// TIA Portal V15.1 export
// export: Created 2020-06-12T07:35:47.7568359Z, ExportSetting None, DisplayName Totally Integrated Automation Portal, DisplayVersion V15.1, DisplayName TIA Portal Openness, DisplayVersion V15.1, DisplayName STEP 7 Professional, DisplayVersion V15.1, DisplayName STEP 7 Safety, DisplayVersion V15.1, DisplayName WinCC Advanced, DisplayVersion V15.1
FUNCTION "DED_unit" : Void   // FC554, FBD
TITLE = Dedusting UNIT
{ S7_Optimized_Access := 'TRUE' }
// stored: SetENOAutomatically False
   VAR_TEMP
      _csf : Bool;   // Common system fault
      tDedOn : Bool;
      tDedOff : Bool;
      tReqOff : Bool;
      tDedDisOn : Bool;
      tDedDisOff : Bool;
      tDisDischTout : Bool;
      tDedDisReqOn1 : Bool;
   END_VAR
   VAR_TEMP   // added for the SCL form of the ladder/FBD networks
      _w1 : Bool;
   END_VAR
BEGIN

REGION Network 1: COMMON SYSTEM FAULT
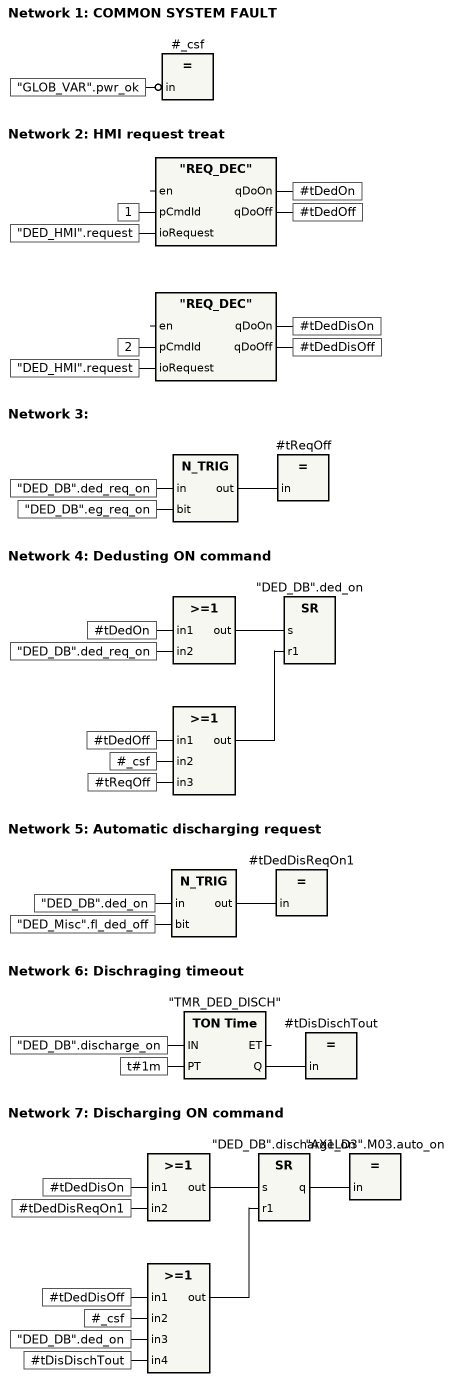
   #_csf := NOT "GLOB_VAR".pwr_ok;
END_REGION

REGION Network 2: HMI request treat
   "REQ_DEC"(pCmdId := 1, ioRequest := "DED_HMI".request, qDoOn => #tDedOn, qDoOff => #tDedOff);
   "REQ_DEC"(pCmdId := 2, ioRequest := "DED_HMI".request, qDoOn => #tDedDisOn, qDoOff => #tDedDisOff);
END_REGION

REGION Network 3
   #_w1 := NOT "DED_DB".ded_req_on AND "DED_DB".eg_req_on;   // falling edge
   "DED_DB".eg_req_on := "DED_DB".ded_req_on;
   #tReqOff := #_w1;
END_REGION

REGION Network 4: Dedusting ON command
   IF #tDedOn OR "DED_DB".ded_req_on THEN
       "DED_DB".ded_on := TRUE;   // SR flip-flop
   END_IF;
   IF #tDedOff OR #_csf OR #tReqOff THEN "DED_DB".ded_on := FALSE; END_IF;
END_REGION

REGION Network 5: Automatic discharging request
   #_w1 := NOT "DED_DB".ded_on AND "DED_Misc".fl_ded_off;   // falling edge
   "DED_Misc".fl_ded_off := "DED_DB".ded_on;
   #tDedDisReqOn1 := #_w1;
END_REGION

REGION Network 6: Dischraging timeout
   "TMR_DED_DISCH".TON(IN := "DED_DB".discharge_on, PT := t#1m);
   #tDisDischTout := "TMR_DED_DISCH".Q;
END_REGION

REGION Network 7: Discharging ON command
   IF #tDedDisOn OR #tDedDisReqOn1 THEN
       "DED_DB".discharge_on := TRUE;   // SR flip-flop
   END_IF;
   IF #tDedDisOff OR #_csf OR "DED_DB".ded_on OR #tDisDischTout THEN "DED_DB".discharge_on := FALSE; END_IF;
   "AX1LD3".M03.auto_on := "DED_DB".discharge_on;
END_REGION

REGION Network 8: Dedusting is running
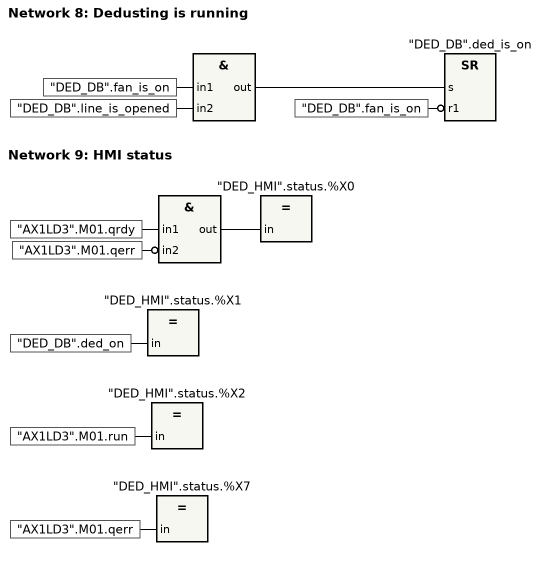
   IF "DED_DB".fan_is_on AND "DED_DB".line_is_opened THEN
       "DED_DB".ded_is_on := TRUE;   // SR flip-flop
   END_IF;
   IF NOT "DED_DB".fan_is_on THEN "DED_DB".ded_is_on := FALSE; END_IF;
END_REGION

REGION Network 9: HMI status
   "DED_HMI".status.%X0 := "AX1LD3".M01.qrdy AND NOT "AX1LD3".M01.qerr;
   "DED_HMI".status.%X1 := "DED_DB".ded_on;
   "DED_HMI".status.%X2 := "AX1LD3".M01.run;
   "DED_HMI".status.%X7 := "AX1LD3".M01.qerr;
END_REGION
END_FUNCTION
